(* Logix 5000 project; controller _2081 vendor 1 type 14 code 77 rev 19.11; software revision 19.01; part 2 of 4 *)
(* tags used below, declared in another part *)
   B23 : DINT[20];   // Fault Bits
   B3 : DINT[10];   // Utility Bits
   B33 : DINT[10];   // Utility Bits
   B36 : DINT[10];   // One-Shots
   F8 : REAL[5];   // Floating Point (Real)
   i1 : INT[8];   // 8-pt Analog Inputs
   i3 : INT;   // Slot 3 16pt DC Input
   i4 : INT;   // Slot 4 16pt DC Input
   N26 : DINT[600];   // Write to PLC
   N27 : DINT[400];   // Read from PLC
   N32 : DINT[200];
   N7 : DINT[250];   // Utility Integers
   o2 : INT[8];   // Slot 2 8-pt Analog Output
   o5 : SINT;   // Slot 5 8-pt Relay Output
   o6 : SINT;   // Slot 6 8-pt Relay Output
   S24 : INT;   // Index Register
   T24 : TIMER[150];   // Fault Timers
   T34 : TIMER[30];   // Utility Timers
   T4 : TIMER[32];
(* BGK_OVEN, continued *)

ROUTINE _02_MAIN   (* ladder *)
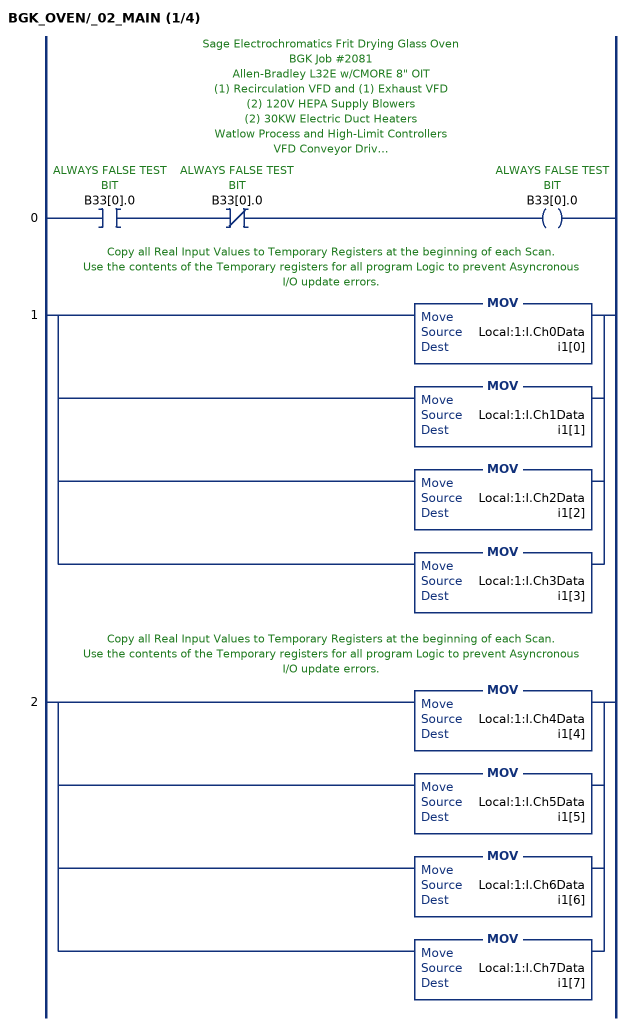
   // Sage Electrochromatics Frit Drying Glass Oven
   // BGK Job #2081
   // Allen-Bradley L32E w/CMORE 8" OIT
   // (1) Recirculation VFD and (1) Exhaust VFD
   // (2) 120V HEPA Supply Blowers
   // (2) 30KW Electric Duct Heaters
   // Watlow Process and High-Limit Controllers
   // VFD Conveyor Drive
   // Lamp Access Lift Motor
   0: XIC(B33[0].0)XIO(B33[0].0)OTE(B33[0].0);
   // Copy all Real Input Values to Temporary Registers at the beginning of each Scan.
   // Use the contents of the Temporary registers for all program Logic to prevent Asyncronous I/O update errors.
   1: [MOV(Local:1:I.Ch0Data,i1[0]) ,MOV(Local:1:I.Ch1Data,i1[1]) ,MOV(Local:1:I.Ch2Data,i1[2]) ,MOV(Local:1:I.Ch3Data,i1[3]) ];
   // Copy all Real Input Values to Temporary Registers at the beginning of each Scan.
   // Use the contents of the Temporary registers for all program Logic to prevent Asyncronous I/O update errors.
   2: [MOV(Local:1:I.Ch4Data,i1[4]) ,MOV(Local:1:I.Ch5Data,i1[5]) ,MOV(Local:1:I.Ch6Data,i1[6]) ,MOV(Local:1:I.Ch7Data,i1[7]) ];
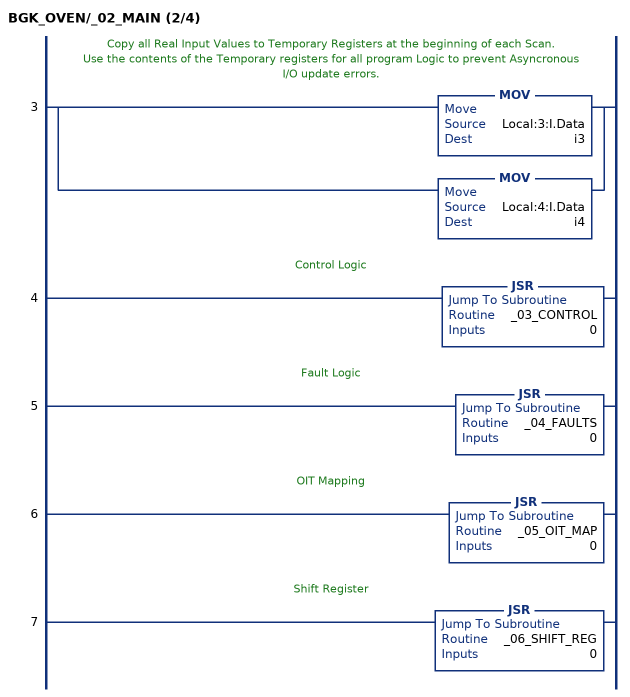
   // Copy all Real Input Values to Temporary Registers at the beginning of each Scan.
   // Use the contents of the Temporary registers for all program Logic to prevent Asyncronous I/O update errors.
   3: [MOV(Local:3:I.Data,i3) ,MOV(Local:4:I.Data,i4) ];
   // Control Logic
   4: JSR(_03_CONTROL,0);
   // Fault Logic
   5: JSR(_04_FAULTS,0);
   // OIT Mapping
   6: JSR(_05_OIT_MAP,0);
   // Shift Register
   7: JSR(_06_SHIFT_REG,0);
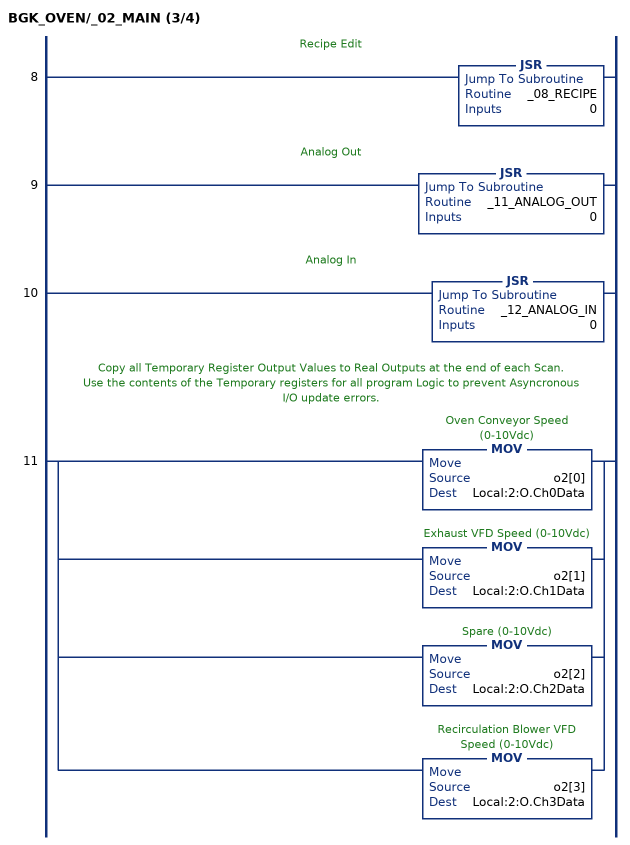
   // Recipe Edit
   8: JSR(_08_RECIPE,0);
   // Analog Out
   9: JSR(_11_ANALOG_OUT,0);
   // Analog In
   10: JSR(_12_ANALOG_IN,0);
   // Copy all Temporary Register Output Values to Real Outputs at the end of each Scan.
   // Use the contents of the Temporary registers for all program Logic to prevent Asyncronous I/O update errors.
   11: [MOV(o2[0],Local:2:O.Ch0Data) ,MOV(o2[1],Local:2:O.Ch1Data) ,MOV(o2[2],Local:2:O.Ch2Data) ,MOV(o2[3],Local:2:O.Ch3Data) ];
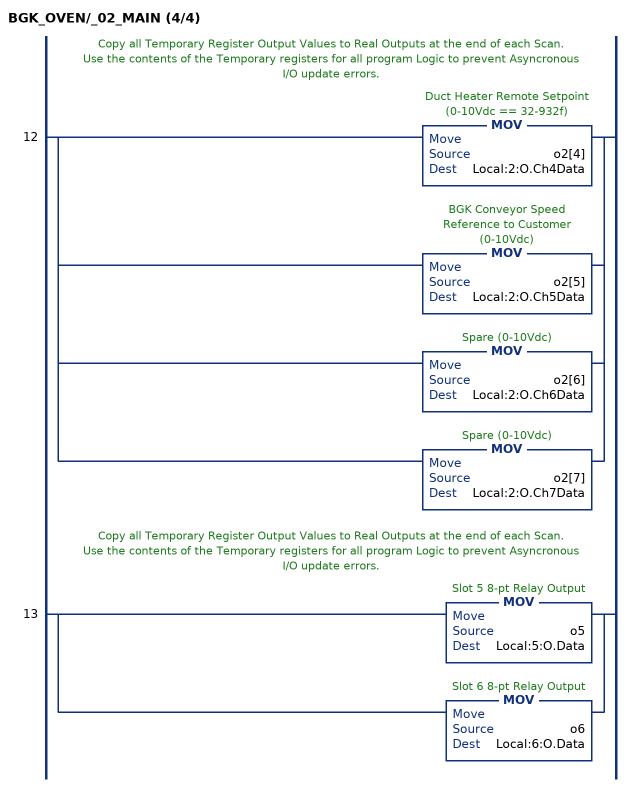
   // Copy all Temporary Register Output Values to Real Outputs at the end of each Scan.
   // Use the contents of the Temporary registers for all program Logic to prevent Asyncronous I/O update errors.
   12: [MOV(o2[4],Local:2:O.Ch4Data) ,MOV(o2[5],Local:2:O.Ch5Data) ,MOV(o2[6],Local:2:O.Ch6Data) ,MOV(o2[7],Local:2:O.Ch7Data) ];
   // Copy all Temporary Register Output Values to Real Outputs at the end of each Scan.
   // Use the contents of the Temporary registers for all program Logic to prevent Asyncronous I/O update errors.
   13: [MOV(o5,Local:5:O.Data) ,MOV(o6,Local:6:O.Data) ];
END_ROUTINE

ROUTINE _03_CONTROL   (* ladder *)
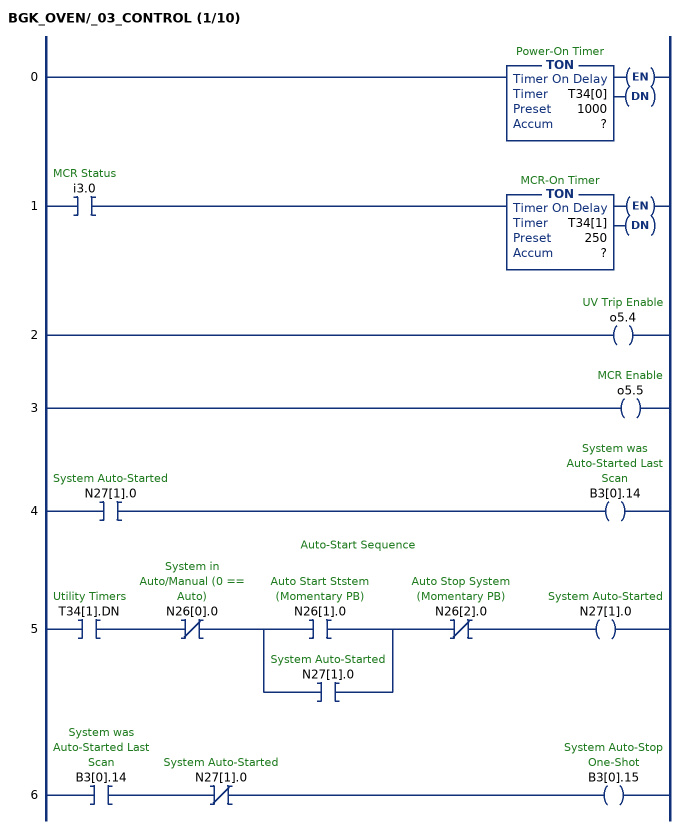
   0: TON(T34[0],?,?);
   1: XIC(i3.0)TON(T34[1],?,?);
   2: OTE(o5.4);
   3: OTE(o5.5);
   4: XIC(N27[1].0)OTE(B3[0].14);
   // Auto-Start Sequence
   5: XIC(T34[1].DN)XIO(N26[0].0)[XIC(N26[1].0) ,XIC(N27[1].0) ]XIO(N26[2].0)OTE(N27[1].0);
   6: XIC(B3[0].14)XIO(N27[1].0)OTE(B3[0].15);
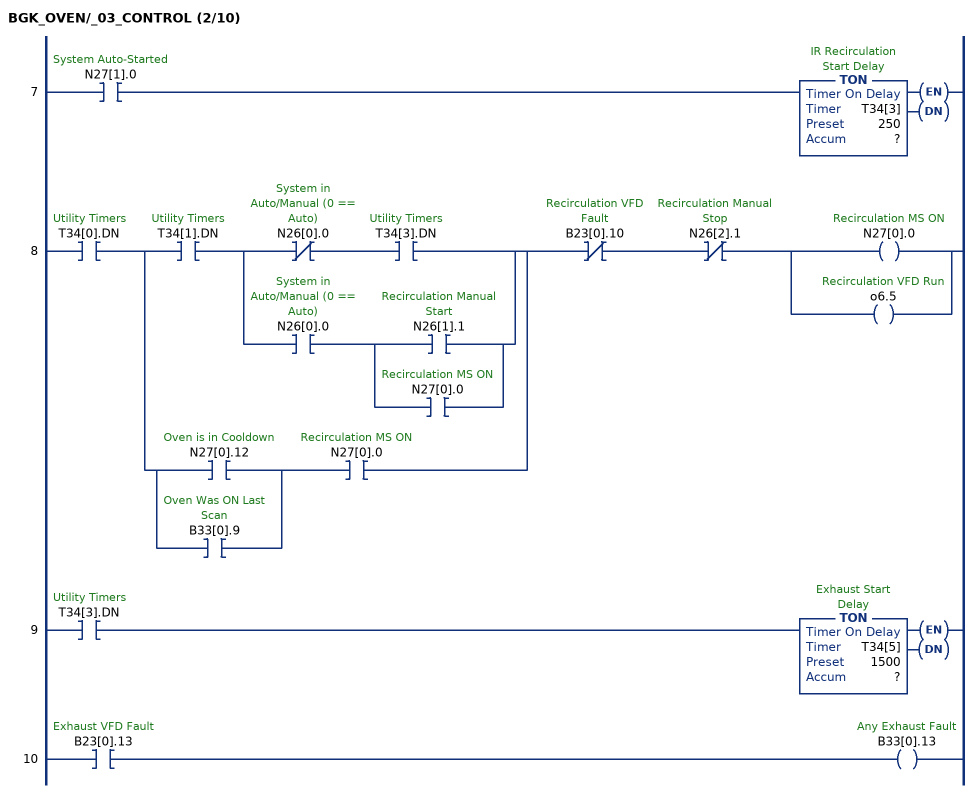
   7: XIC(N27[1].0)TON(T34[3],?,?);
   8: XIC(T34[0].DN)[XIC(T34[1].DN) [XIO(N26[0].0) XIC(T34[3].DN) ,XIC(N26[0].0) [XIC(N26[1].1) ,XIC(N27[0].0) ] ] ,[XIC(N27[0].12) ,XIC(B33[0].9) ] XIC(N27[0].0) ]XIO(B23[0].10)XIO(N26[2].1)[OTE(N27[0].0) ,OTE(o6.5) ];
   9: XIC(T34[3].DN)TON(T34[5],?,?);
   10: XIC(B23[0].13)OTE(B33[0].13);
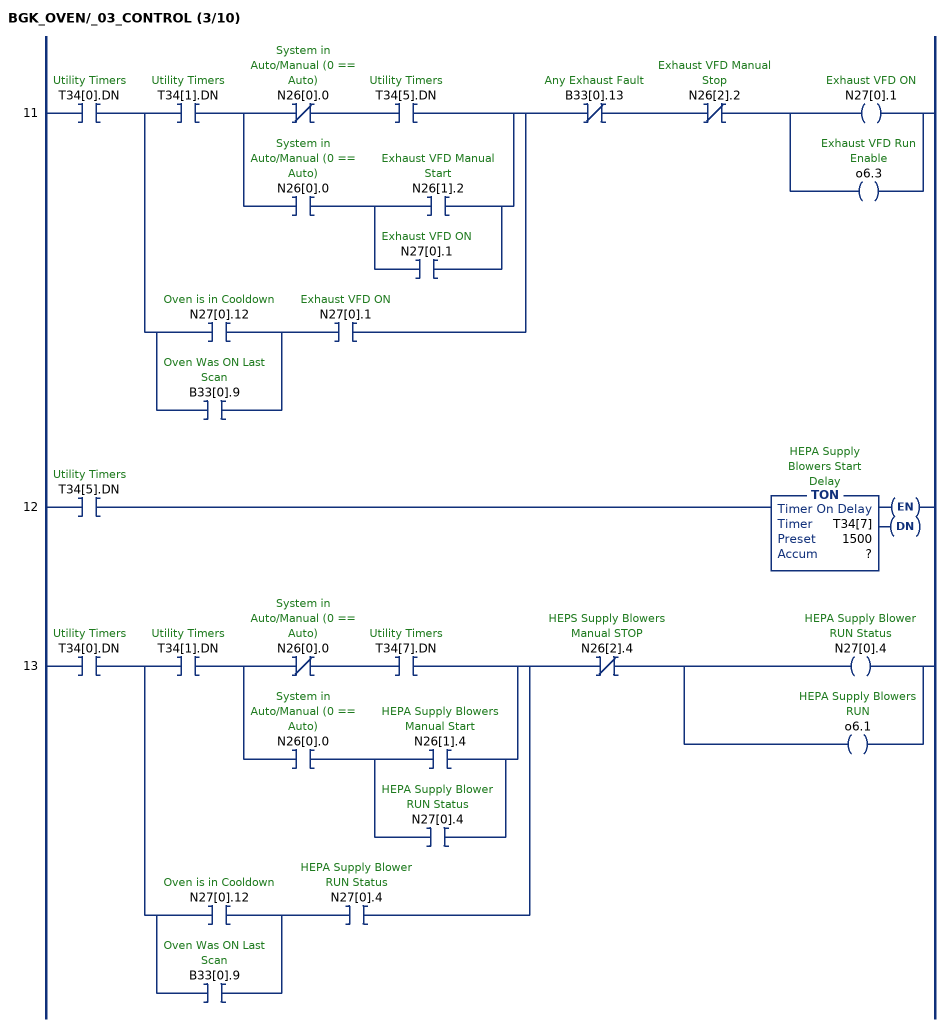
   11: XIC(T34[0].DN)[XIC(T34[1].DN) [XIO(N26[0].0) XIC(T34[5].DN) ,XIC(N26[0].0) [XIC(N26[1].2) ,XIC(N27[0].1) ] ] ,[XIC(N27[0].12) ,XIC(B33[0].9) ] XIC(N27[0].1) ]XIO(B33[0].13)XIO(N26[2].2)[OTE(N27[0].1) ,OTE(o6.3) ];
   12: XIC(T34[5].DN)TON(T34[7],?,?);
   13: XIC(T34[0].DN)[XIC(T34[1].DN) [XIO(N26[0].0) XIC(T34[7].DN) ,XIC(N26[0].0) [XIC(N26[1].4) ,XIC(N27[0].4) ] ] ,[XIC(N27[0].12) ,XIC(B33[0].9) ] XIC(N27[0].4) ]XIO(N26[2].4)[OTE(N27[0].4) ,OTE(o6.1) ];
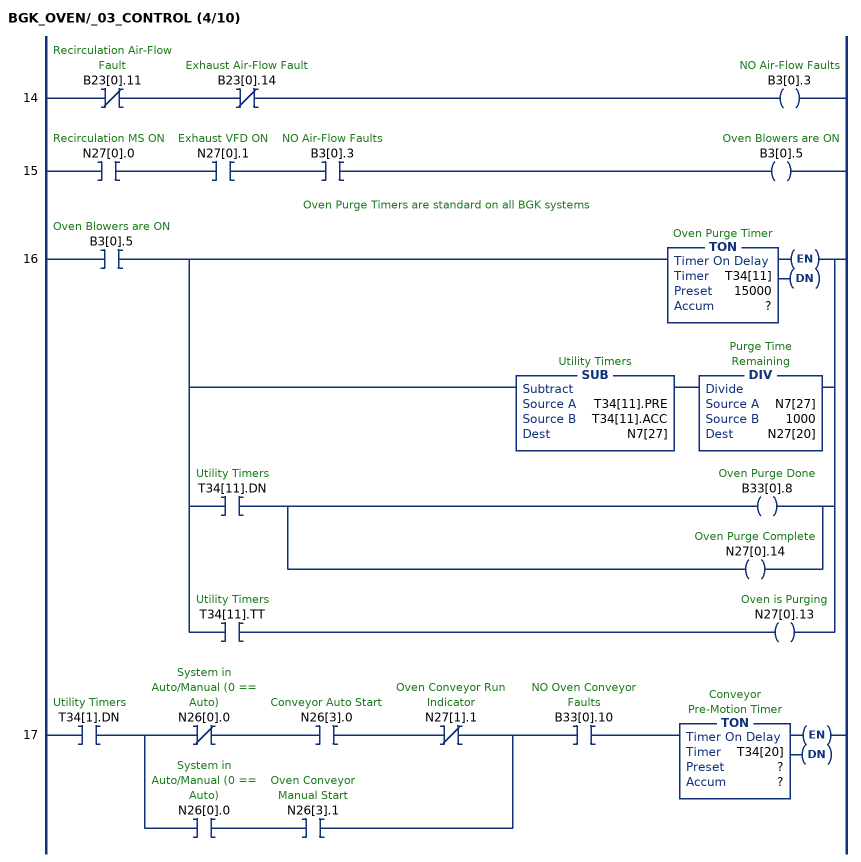
   14: XIO(B23[0].11)XIO(B23[0].14)OTE(B3[0].3);
   15: XIC(N27[0].0)XIC(N27[0].1)XIC(B3[0].3)OTE(B3[0].5);
   // Oven Purge Timers are standard on all BGK systems
   16: XIC(B3[0].5)[TON(T34[11],?,?) ,SUB(T34[11].PRE,T34[11].ACC,N7[27]) DIV(N7[27],1000,N27[20]) ,XIC(T34[11].DN) [OTE(B33[0].8) ,OTE(N27[0].14) ] ,XIC(T34[11].TT) OTE(N27[0].13) ];
   17: XIC(T34[1].DN)[XIO(N26[0].0) XIC(N26[3].0) XIO(N27[1].1) ,XIC(N26[0].0) XIC(N26[3].1) ]XIC(B33[0].10)TON(T34[20],?,?);
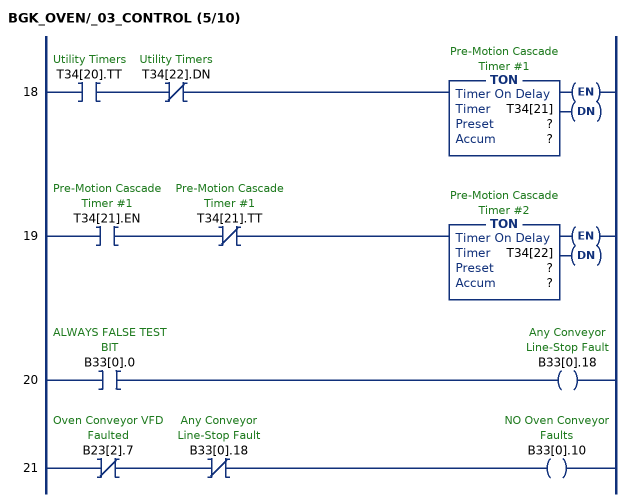
   18: XIC(T34[20].TT)XIO(T34[22].DN)TON(T34[21],?,?);
   19: XIC(T34[21].EN)XIO(T34[21].TT)TON(T34[22],?,?);
   20: XIC(B33[0].0)OTE(B33[0].18);
   21: XIO(B23[2].7)XIO(B33[0].18)OTE(B33[0].10);
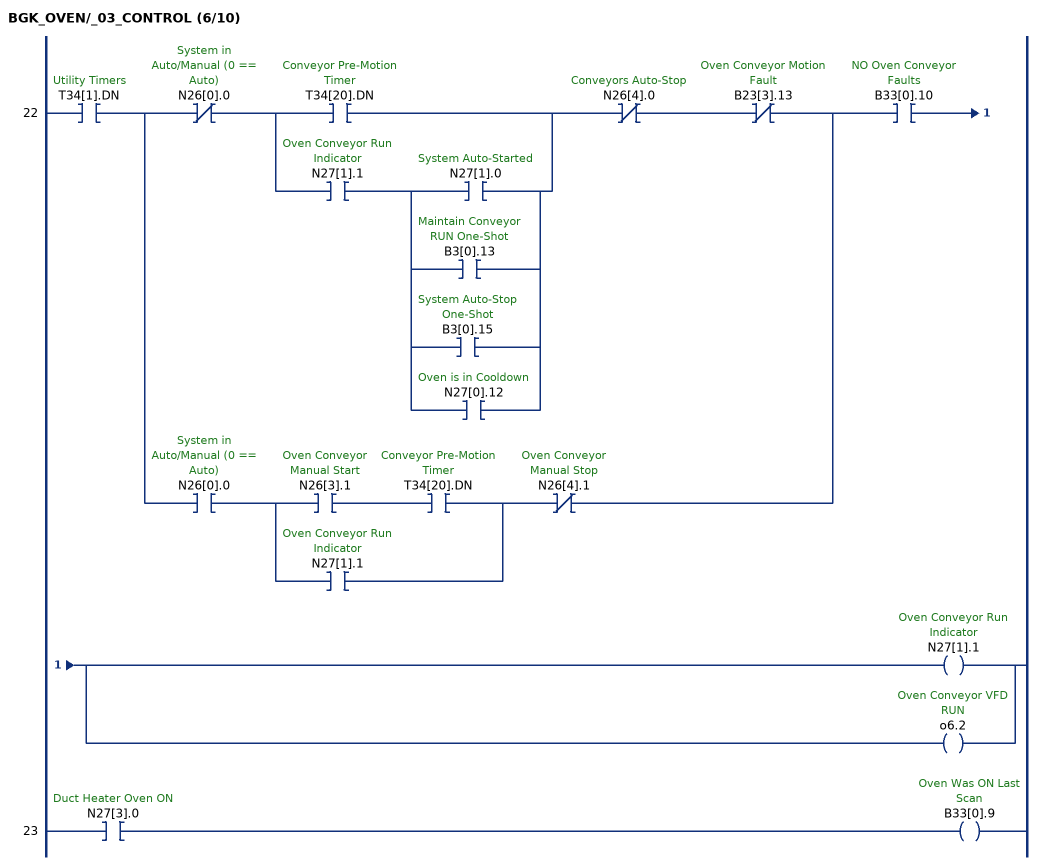
   22: XIC(T34[1].DN)[XIO(N26[0].0) [XIC(T34[20].DN) ,XIC(N27[1].1) [XIC(N27[1].0) ,XIC(B3[0].13) ,XIC(B3[0].15) ,XIC(N27[0].12) ] ] XIO(N26[4].0) XIO(B23[3].13) ,XIC(N26[0].0) [XIC(N26[3].1) XIC(T34[20].DN) ,XIC(N27[1].1) ] XIO(N26[4].1) ]XIC(B33[0].10)[OTE(N27[1].1) ,OTE(o6.2) ];
   23: XIC(N27[3].0)OTE(B33[0].9);
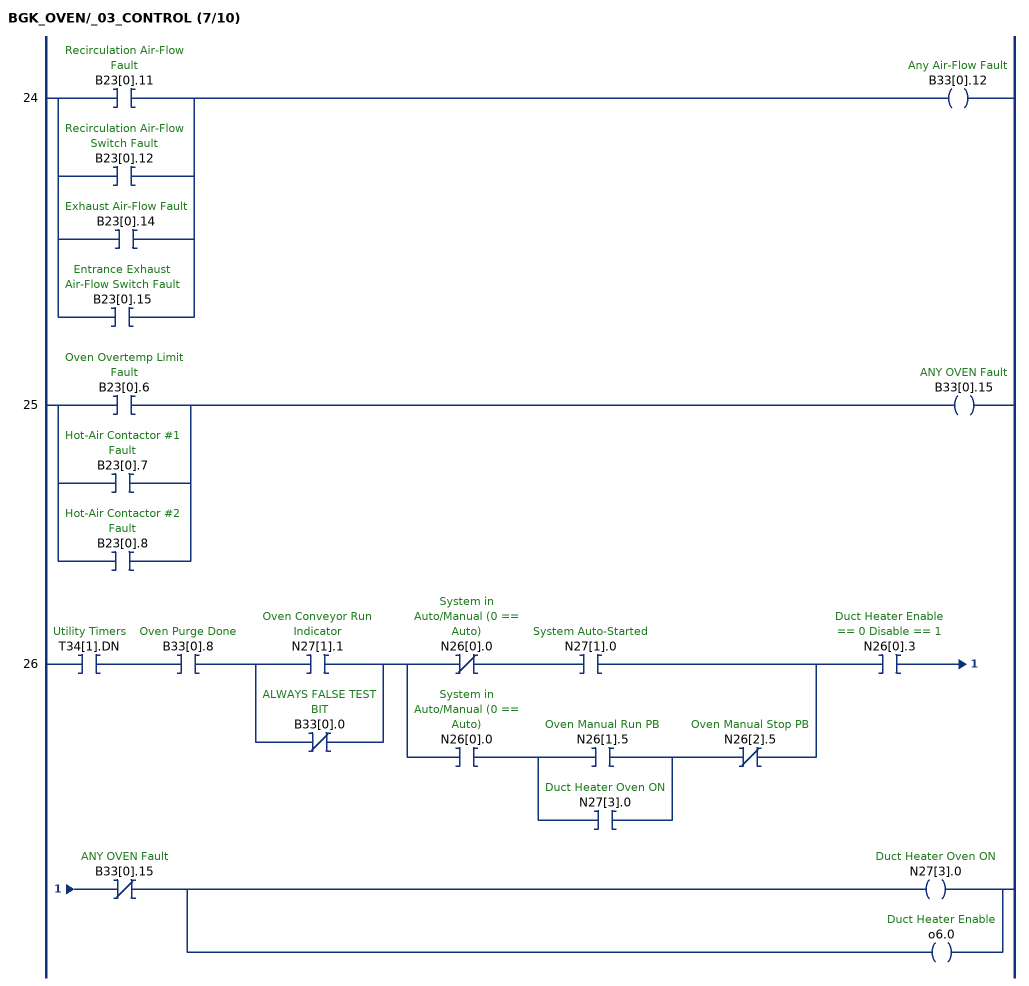
   24: [XIC(B23[0].11) ,XIC(B23[0].12) ,XIC(B23[0].14) ,XIC(B23[0].15) ]OTE(B33[0].12);
   25: [XIC(B23[0].6) ,XIC(B23[0].7) ,XIC(B23[0].8) ]OTE(B33[0].15);
   26: XIC(T34[1].DN)XIC(B33[0].8)[XIC(N27[1].1) ,XIO(B33[0].0) ][XIO(N26[0].0) XIC(N27[1].0) ,XIC(N26[0].0) [XIC(N26[1].5) ,XIC(N27[3].0) ] XIO(N26[2].5) ]XIC(N26[0].3)XIO(B33[0].15)[OTE(N27[3].0) ,OTE(o6.0) ];
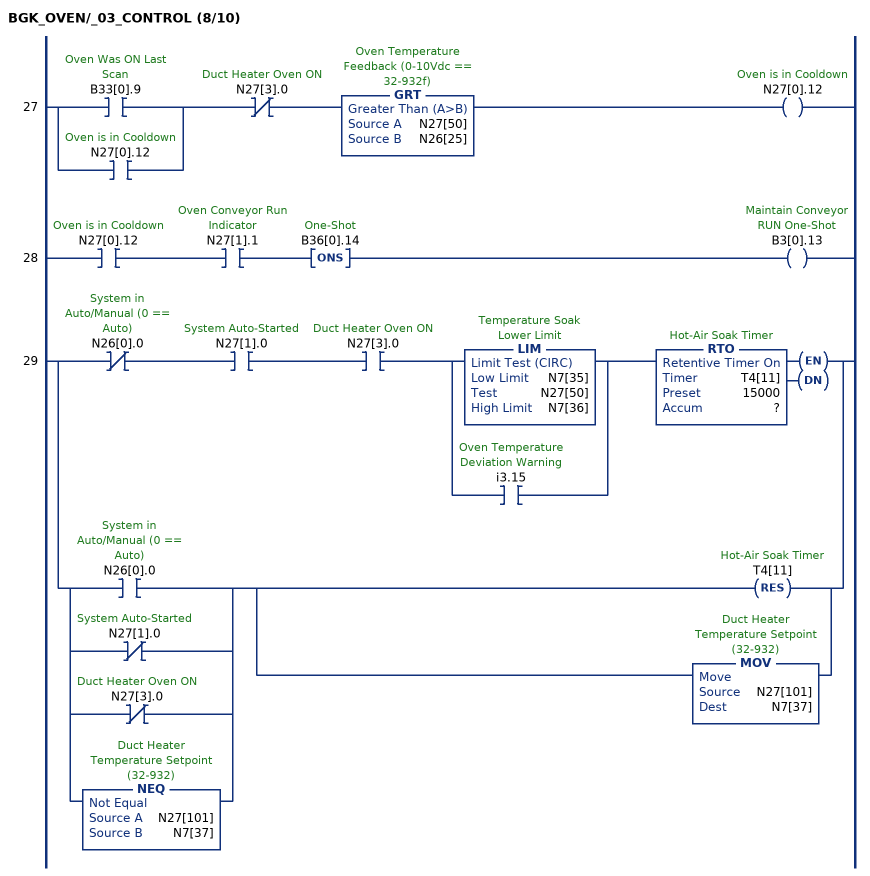
   27: [XIC(B33[0].9) ,XIC(N27[0].12) ]XIO(N27[3].0)GRT(N27[50],N26[25])OTE(N27[0].12);
   28: XIC(N27[0].12)XIC(N27[1].1)ONS(B36[0].14)OTE(B3[0].13);
   29: [XIO(N26[0].0) XIC(N27[1].0) XIC(N27[3].0) [LIM(N7[35],N27[50],N7[36]) ,XIC(i3.15) ] RTO(T4[11],?,?) ,[XIC(N26[0].0) ,XIO(N27[1].0) ,XIO(N27[3].0) ,NEQ(N27[101],N7[37]) ] [RES(T4[11]) ,MOV(N27[101],N7[37]) ] ];
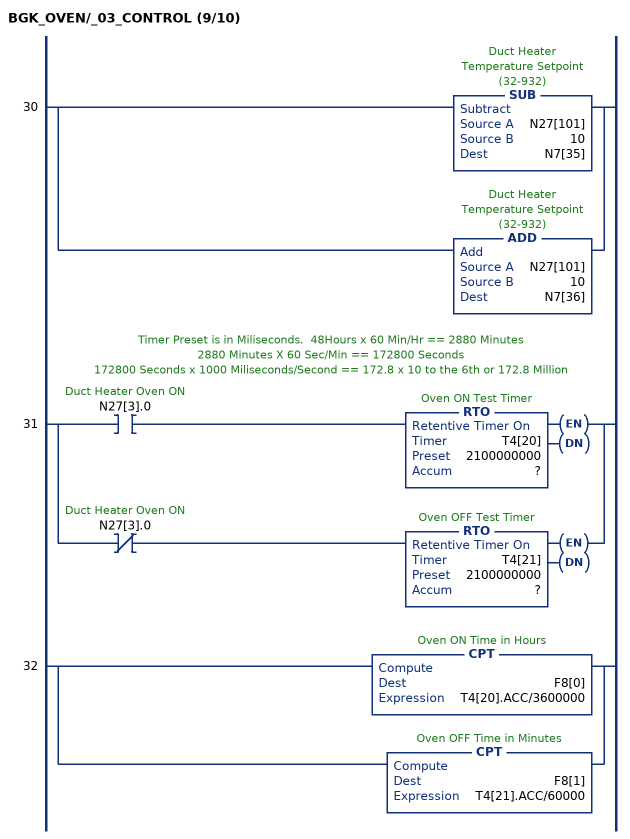
   30: [SUB(N27[101],10,N7[35]) ,ADD(N27[101],10,N7[36]) ];
   // Timer Preset is in Miliseconds.  48Hours x 60 Min/Hr == 2880 Minutes
   // 2880 Minutes X 60 Sec/Min == 172800 Seconds
   // 172800 Seconds x 1000 Miliseconds/Second == 172.8 x 10 to the 6th or 172.8 Million
   31: [XIC(N27[3].0) RTO(T4[20],?,?) ,XIO(N27[3].0) RTO(T4[21],?,?) ];
   32: [CPT(F8[0],T4[20].ACC/3600000) ,CPT(F8[1],T4[21].ACC/60000) ];
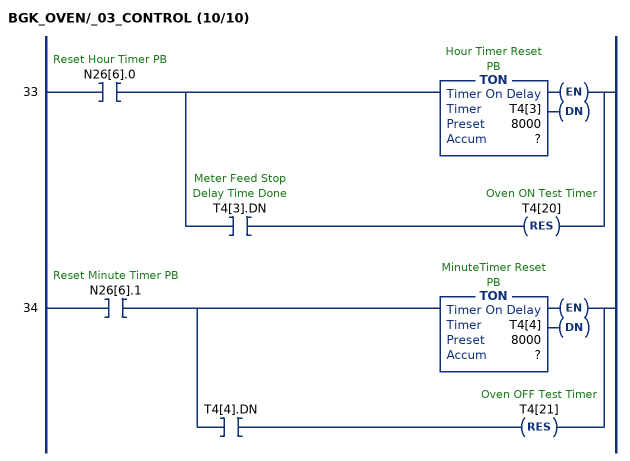
   33: XIC(N26[6].0)[TON(T4[3],?,?) ,XIC(T4[3].DN) RES(T4[20]) ];
   34: XIC(N26[6].1)[TON(T4[4],?,?) ,XIC(T4[4].DN) RES(T4[21]) ];
END_ROUTINE

ROUTINE _04_FAULTS   (* ladder *)
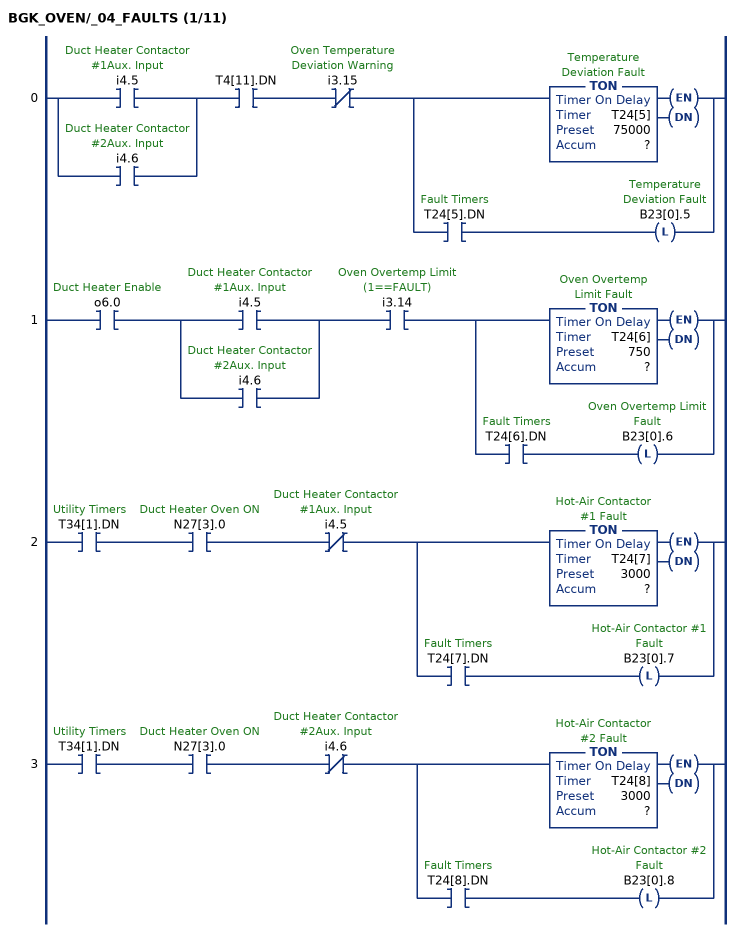
   0: [XIC(i4.5) ,XIC(i4.6) ]XIC(T4[11].DN)XIO(i3.15)[TON(T24[5],?,?) ,XIC(T24[5].DN) OTL(B23[0].5) ];
   1: XIC(o6.0)[XIC(i4.5) ,XIC(i4.6) ]XIC(i3.14)[TON(T24[6],?,?) ,XIC(T24[6].DN) OTL(B23[0].6) ];
   2: XIC(T34[1].DN)XIC(N27[3].0)XIO(i4.5)[TON(T24[7],?,?) ,XIC(T24[7].DN) OTL(B23[0].7) ];
   3: XIC(T34[1].DN)XIC(N27[3].0)XIO(i4.6)[TON(T24[8],?,?) ,XIC(T24[8].DN) OTL(B23[0].8) ];
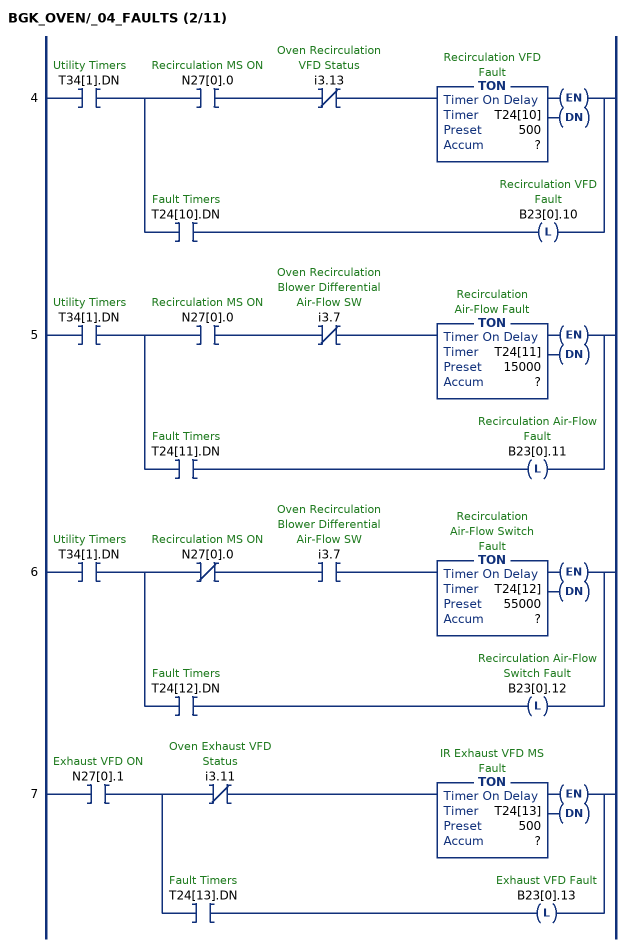
   4: XIC(T34[1].DN)[XIC(N27[0].0) XIO(i3.13) TON(T24[10],?,?) ,XIC(T24[10].DN) OTL(B23[0].10) ];
   5: XIC(T34[1].DN)[XIC(N27[0].0) XIO(i3.7) TON(T24[11],?,?) ,XIC(T24[11].DN) OTL(B23[0].11) ];
   6: XIC(T34[1].DN)[XIO(N27[0].0) XIC(i3.7) TON(T24[12],?,?) ,XIC(T24[12].DN) OTL(B23[0].12) ];
   7: XIC(N27[0].1)[XIO(i3.11) TON(T24[13],?,?) ,XIC(T24[13].DN) OTL(B23[0].13) ];
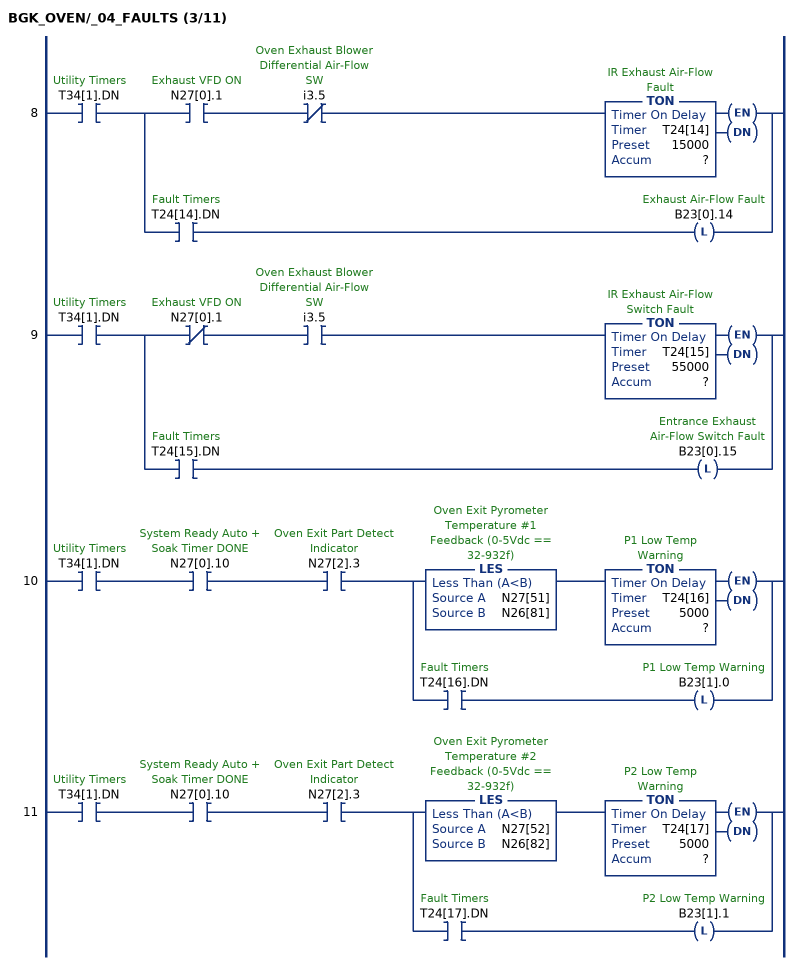
   8: XIC(T34[1].DN)[XIC(N27[0].1) XIO(i3.5) TON(T24[14],?,?) ,XIC(T24[14].DN) OTL(B23[0].14) ];
   9: XIC(T34[1].DN)[XIO(N27[0].1) XIC(i3.5) TON(T24[15],?,?) ,XIC(T24[15].DN) OTL(B23[0].15) ];
   10: XIC(T34[1].DN)XIC(N27[0].10)XIC(N27[2].3)[LES(N27[51],N26[81]) TON(T24[16],?,?) ,XIC(T24[16].DN) OTL(B23[1].0) ];
   11: XIC(T34[1].DN)XIC(N27[0].10)XIC(N27[2].3)[LES(N27[52],N26[82]) TON(T24[17],?,?) ,XIC(T24[17].DN) OTL(B23[1].1) ];
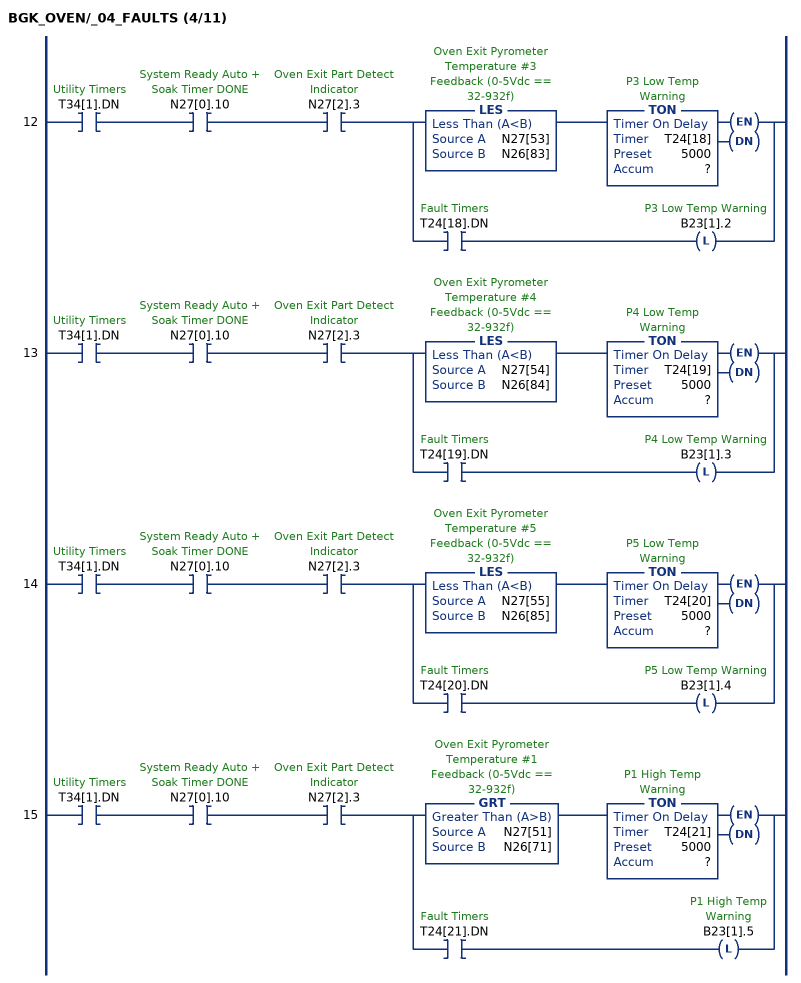
   12: XIC(T34[1].DN)XIC(N27[0].10)XIC(N27[2].3)[LES(N27[53],N26[83]) TON(T24[18],?,?) ,XIC(T24[18].DN) OTL(B23[1].2) ];
   13: XIC(T34[1].DN)XIC(N27[0].10)XIC(N27[2].3)[LES(N27[54],N26[84]) TON(T24[19],?,?) ,XIC(T24[19].DN) OTL(B23[1].3) ];
   14: XIC(T34[1].DN)XIC(N27[0].10)XIC(N27[2].3)[LES(N27[55],N26[85]) TON(T24[20],?,?) ,XIC(T24[20].DN) OTL(B23[1].4) ];
   15: XIC(T34[1].DN)XIC(N27[0].10)XIC(N27[2].3)[GRT(N27[51],N26[71]) TON(T24[21],?,?) ,XIC(T24[21].DN) OTL(B23[1].5) ];
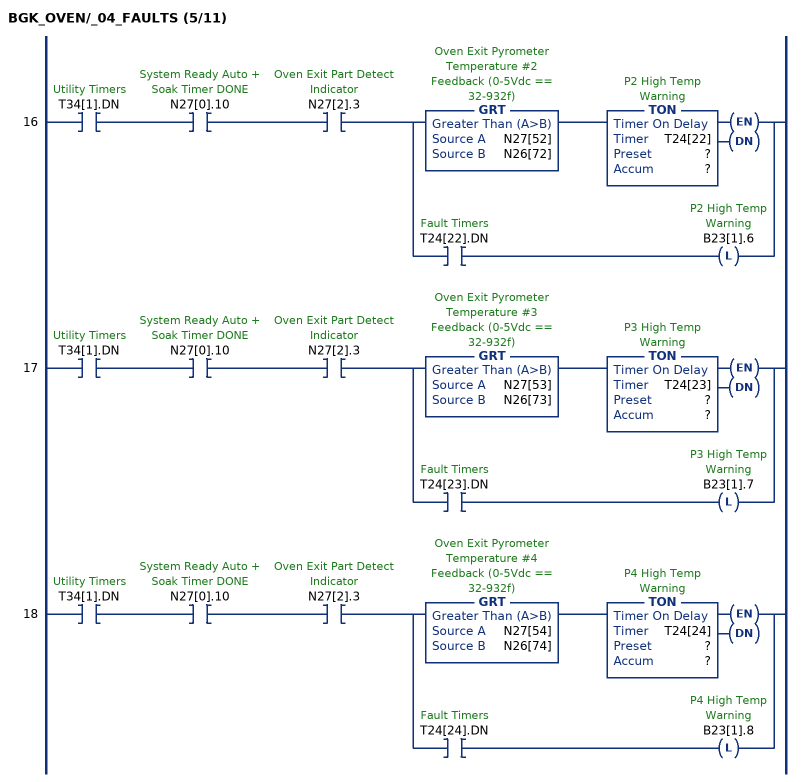
   16: XIC(T34[1].DN)XIC(N27[0].10)XIC(N27[2].3)[GRT(N27[52],N26[72]) TON(T24[22],?,?) ,XIC(T24[22].DN) OTL(B23[1].6) ];
   17: XIC(T34[1].DN)XIC(N27[0].10)XIC(N27[2].3)[GRT(N27[53],N26[73]) TON(T24[23],?,?) ,XIC(T24[23].DN) OTL(B23[1].7) ];
   18: XIC(T34[1].DN)XIC(N27[0].10)XIC(N27[2].3)[GRT(N27[54],N26[74]) TON(T24[24],?,?) ,XIC(T24[24].DN) OTL(B23[1].8) ];
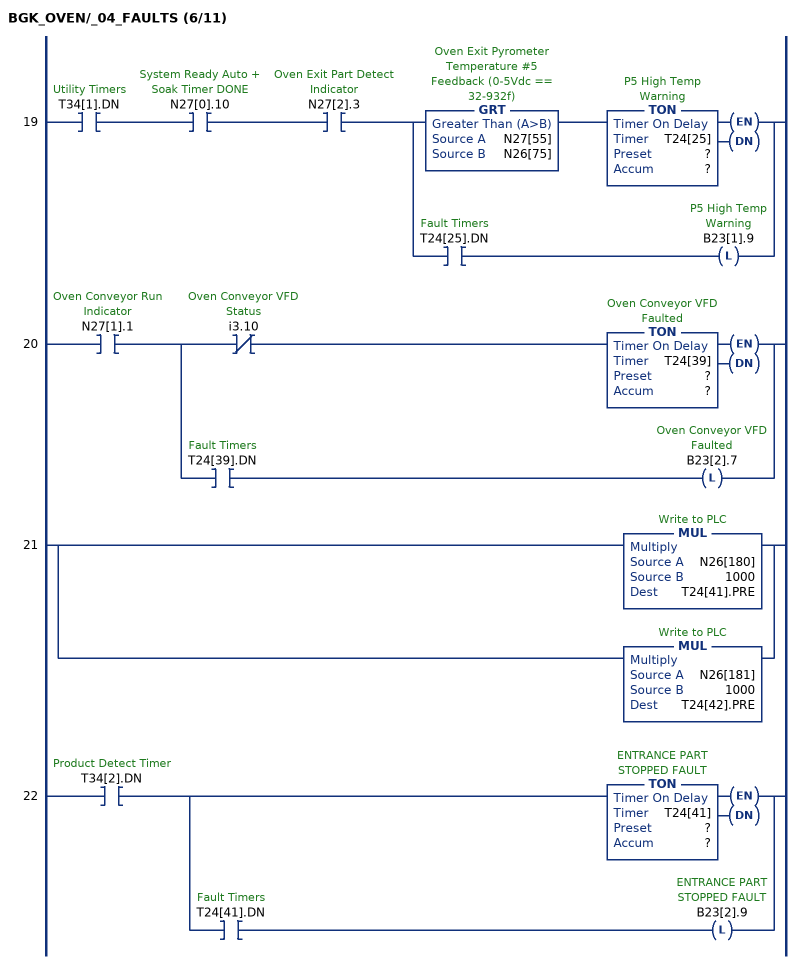
   19: XIC(T34[1].DN)XIC(N27[0].10)XIC(N27[2].3)[GRT(N27[55],N26[75]) TON(T24[25],?,?) ,XIC(T24[25].DN) OTL(B23[1].9) ];
   20: XIC(N27[1].1)[XIO(i3.10) TON(T24[39],?,?) ,XIC(T24[39].DN) OTL(B23[2].7) ];
   21: [MUL(N26[180],1000,T24[41].PRE) ,MUL(N26[181],1000,T24[42].PRE) ];
   22: XIC(T34[2].DN)[TON(T24[41],?,?) ,XIC(T24[41].DN) OTL(B23[2].9) ];
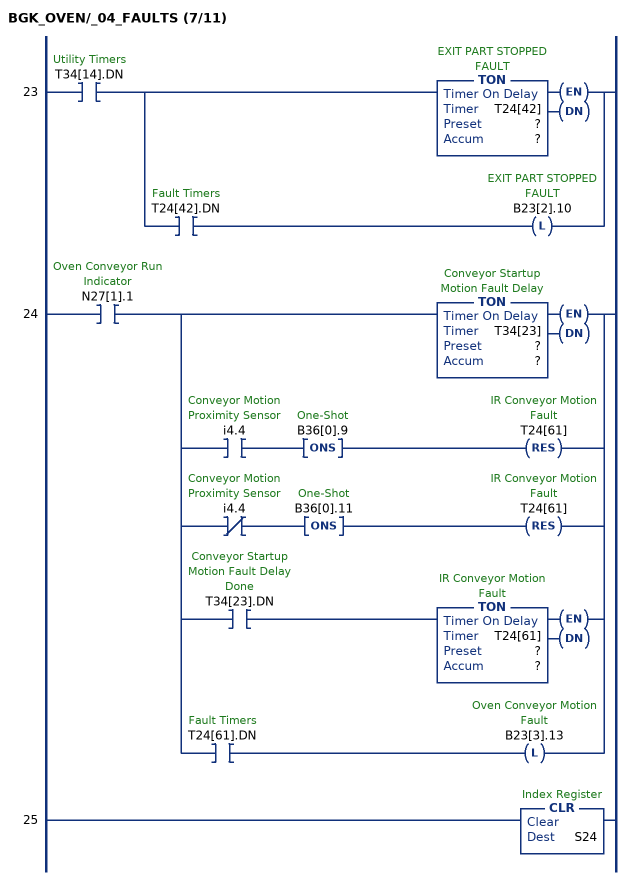
   23: XIC(T34[14].DN)[TON(T24[42],?,?) ,XIC(T24[42].DN) OTL(B23[2].10) ];
   24: XIC(N27[1].1)[TON(T34[23],?,?) ,XIC(i4.4) ONS(B36[0].9) RES(T24[61]) ,XIO(i4.4) ONS(B36[0].11) RES(T24[61]) ,XIC(T34[23].DN) TON(T24[61],?,?) ,XIC(T24[61].DN) OTL(B23[3].13) ];
   25: CLR(S24);
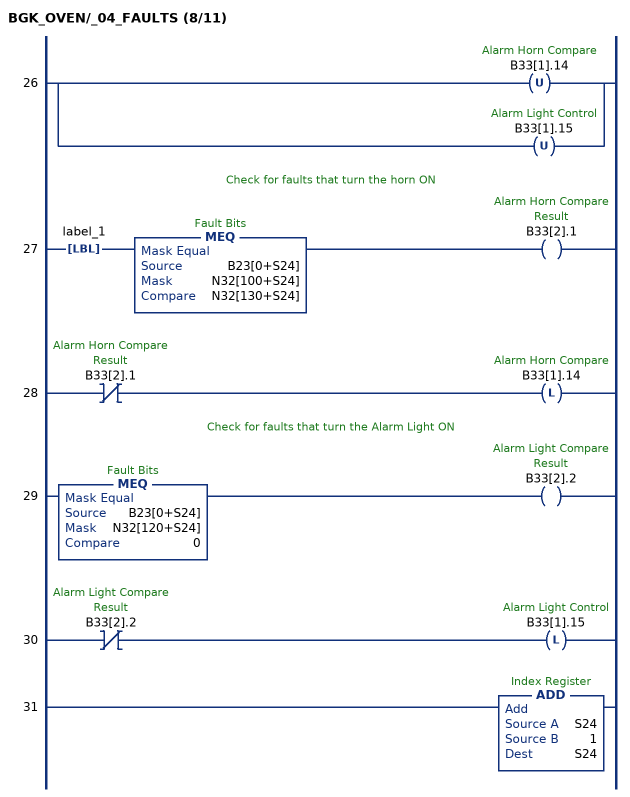
   26: [OTU(B33[1].14) ,OTU(B33[1].15) ];
   // Check for faults that turn the horn ON
   27: LBL(label_1)MEQ(B23[0+S24],N32[100+S24],N32[130+S24])OTE(B33[2].1);
   28: XIO(B33[2].1)OTL(B33[1].14);
   // Check for faults that turn the Alarm Light ON
   29: MEQ(B23[0+S24],N32[120+S24],0)OTE(B33[2].2);
   30: XIO(B33[2].2)OTL(B33[1].15);
   31: ADD(S24,1,S24);
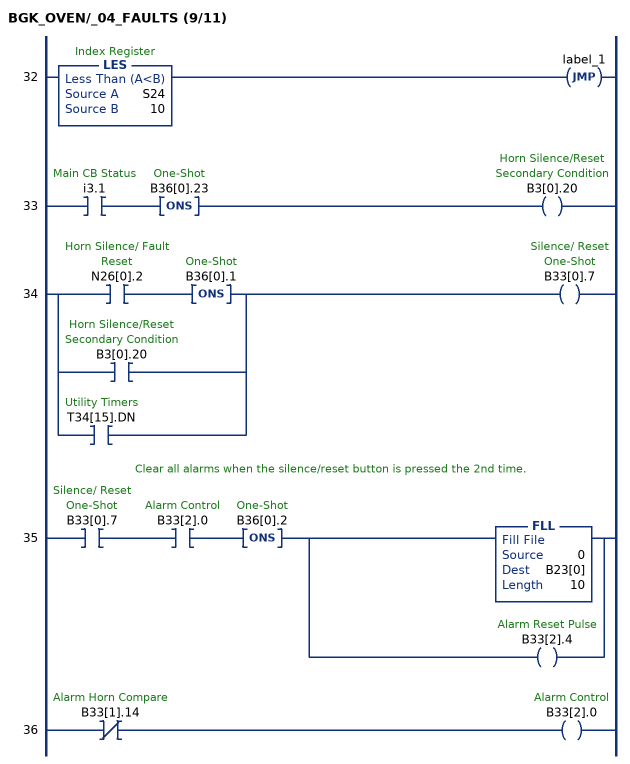
   32: LES(S24,10)JMP(label_1);
   33: XIC(i3.1)ONS(B36[0].23)OTE(B3[0].20);
   34: [XIC(N26[0].2) ONS(B36[0].1) ,XIC(B3[0].20) ,XIC(T34[15].DN) ]OTE(B33[0].7);
   // Clear all alarms when the silence/reset button is pressed the 2nd time.
   35: XIC(B33[0].7)XIC(B33[2].0)ONS(B36[0].2)[FLL(0,B23[0],10) ,OTE(B33[2].4) ];
   36: XIO(B33[1].14)OTE(B33[2].0);
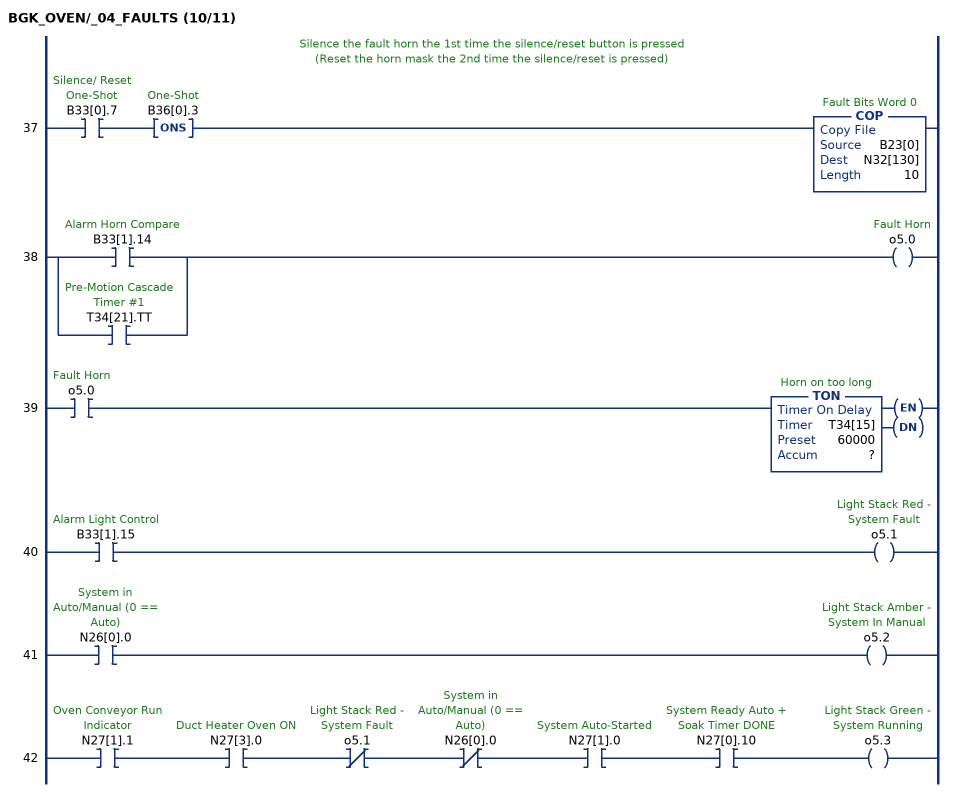
   // Silence the fault horn the 1st time the silence/reset button is pressed
   // (Reset the horn mask the 2nd time the silence/reset is pressed)
   37: XIC(B33[0].7)ONS(B36[0].3)COP(B23[0],N32[130],10);
   38: [XIC(B33[1].14) ,XIC(T34[21].TT) ]OTE(o5.0);
   39: XIC(o5.0)TON(T34[15],?,?);
   40: XIC(B33[1].15)OTE(o5.1);
   41: XIC(N26[0].0)OTE(o5.2);
   42: XIC(N27[1].1)XIC(N27[3].0)XIO(o5.1)XIO(N26[0].0)XIC(N27[1].0)XIC(N27[0].10)OTE(o5.3);
